PROGRAM RESTFUL_API
VAR
    bPostPushover : BOOL;
    fbHttpClientPushover        : FB_IotHttpClient :=(sHostName:='api.pushover.net',
                                     bKeepAlive:=TRUE, tConnectionTimeout:=T#10S);
    fbHttpPostPushover            : FB_Pushover;
	sMyToken               		   : STRING(30) := 'azggdmmagry5dgeskpoj2m8tgrk4w2';
	sMyUser				 		   : STRING(30) := 'uaeadvuczqtdh4dftqornb8i5cn79e';
	sMyMessage			 		   : STRING(180);
	sMyDevice				 	   : STRING(20) ;
	sMyTitle				       : STRING(20);
	
END_VAR

//init client parameters at startup
IF NOT fbHttpClientPushover.bConfigured THEN
    fbHttpClientPushover.nHostPort:= 80;
    fbHttpClientPushover.stTLS.bNoServerCertCheck:= FALSE;
END_IF

IF fbHttpClientPushover.bConfigured THEN
    fbHttpPostPushover(bSend:=bPostPushover, fbClient:=fbHttpClientPushover, sToken := sMyToken, sUser := sMyUser, sMessage :=sMyMessage, sDevice := sMyDevice, sTitle:= sMyTitle, iPriority := -1 );
END_IF

fbHttpClientPushover.Execute();

END_PROGRAM

(* stored: Version 1.1.0.1, ProductVersion 3.1.4024.13
   POU RESTFUL_API: Id {f476f757-ca2c-4df2-9470-6a492022d4f9}, SpecialFunc None *)
